FUNCTION F_AddMessage : BOOL
VAR_IN_OUT
	Station	: Station;
END_VAR

VAR_INPUT
	Text		: T_MaxString;
	AltText		: T_MaxString;
	Color		: DINT;
	Channel		: DINT;
END_VAR

VAR
	HMIMessage		: HMIMessage;
END_VAR

// Construct HMI Message
HMIMessage.Text 	:= Text;
HMIMessage.AltText 	:= AltText;
HMIMessage.Color 	:= Color;
HMIMessage.Channel 	:= Channel;

// Load HMI Message to Station FIFO
Station.HMIMessageFIFO.LOAD(pFIFO := ADR(Station.HMIMessageBuffer), in := HMIMessage);

END_FUNCTION

(* stored: Version 1.1.0.1, ProductVersion 3.1.4024.9
   POU F_AddMessage: Id {57825879-dd46-4c12-a392-0ad38417e32d}, SpecialFunc None *)
